Yaskawa INFORM job: FRONT_WELD_0ST-2_4640.JBI

/JOB
//NAME FRONT_WELD_0ST-2_4640
///FOLDERNAME 02-SKRZYNIE_JOBS
//POS
///NPOS 115,115,0,17,0,0
///TOOL 0
///POSTYPE PULSE
///PULSE
C00000=1212,-39190,49707,1936,-15809,-581
C00001=-55064,-17017,13106,20113,45767,-35735
C00002=-85641,-3161,12660,31281,67420,-55579
C00003=-77611,9747,38455,32702,57795,-55547
C00004=-77611,9747,38455,32702,57795,-55547
C00005=-80481,23547,61641,37204,60115,-56891
C00006=-80479,11681,28780,33754,71138,-52780
C00007=-73572,15026,34389,33675,67405,-51294
C00008=-73572,19926,48501,35202,62492,-53068
C00009=-82806,26311,53816,38180,73291,-53604
C00010=-71695,3747,16001,30713,64750,-51022
C00011=-70421,5575,20105,30867,63066,-51036
C00012=-35543,-20105,-5144,22821,50284,-40173
C00013=-37830,-23193,-8618,23571,50957,-40982
C00014=11136,-28839,-12562,1025,41780,-20887
C00015=20486,-27077,-7346,-12554,38415,-10736
C00016=59545,-9921,5571,-27063,51925,3267
C00017=55110,-17412,-5825,-19778,50988,-2825
C00018=79390,11759,28162,-35512,71262,52960
C00019=74811,13878,33986,-35807,67493,52464
C00020=74942,18762,48004,-37392,62815,54352
C00021=76815,18630,46530,-37158,64288,54543
C00022=79390,11759,28162,-35512,71262,52960
C00023=10831,-54278,-29128,-6468,39852,-5090
C00024=-67200,-10549,24402,-3189,24913,-39001
C00025=-75122,-2194,12822,3152,39225,-43427
C00026=-77516,10189,32861,8493,33365,-45533
C00027=-75154,17575,49272,7885,27457,-44928
C00028=-68113,9932,38901,1157,28472,-40453
C00029=-67114,5383,31515,9208,32648,-43213
C00030=-66450,3998,29285,10896,33890,-43630
C00031=-66374,3101,28136,14657,35566,-44954
C00032=-66747,-26,23691,26916,43760,-49061
C00033=-69992,3685,29239,35234,50920,-52492
C00034=-77050,-3138,8526,33226,61087,-51698
C00035=-67200,-10549,24402,-3189,24913,-39001
C00036=0,-52280,40443,83103,28146,-16510
C00037=99993,-20782,22705,-13349,24734,56519
C00038=67200,-10549,24402,3189,24913,39001
C00039=75122,-2194,12822,-3152,39225,43427
C00040=74323,5203,27259,-5972,33194,43789
C00041=74015,16414,48063,-6821,27325,44224
C00042=56519,1138,28747,9235,29393,33453
C00043=55467,619,28251,10155,29461,32830
C00044=56374,-724,25854,4078,30541,35419
C00045=56354,-7060,16047,-17622,38436,43274
C00046=68252,956,25699,-34035,49810,51639
C00047=77050,-3138,8526,-33226,61087,51698
C00048=67200,-10549,24402,3189,24913,39001
C00049=0,-52280,40443,-83103,28146,16510
C00050=-99993,-20782,22705,13349,24734,-56519
C00051=-91125,453,39555,30378,52425,-51131
C00052=-81425,-5449,14825,37552,56592,-47667
C00053=-81425,-10835,-2515,34915,62871,-45127
C00054=-79239,4305,16082,37593,68846,-50182
C00055=-81302,5892,27588,46359,62943,-54679
C00056=-82227,19402,59913,51524,57300,-60581
C00057=-84844,8890,27031,38640,69740,-53449
C00058=-90096,4679,14083,37467,76581,-51973
C00059=-87885,29238,52923,40761,81198,69685
C00060=-84355,23847,39024,40698,83720,72224
C00061=-81960,27335,46957,41070,80536,71891
C00062=-82643,24718,50492,48951,72637,70260
C00063=-90480,18737,31939,47254,81986,71631
C00064=-94217,10634,17426,46901,86469,-59967
C00065=-81425,-10835,-2515,34915,62871,-45127
C00066=-81425,-5449,14825,37552,56592,-47667
C00067=-94290,-610,44819,32366,49686,-53459
C00068=0,-55136,17047,60468,32096,-4233
C00069=99993,-20782,22705,-13349,24734,56519
C00070=91125,453,39555,-30378,52425,51131
C00071=81425,-5449,14825,-37552,56592,47667
C00072=81425,-10835,-2515,-34915,62871,45127
C00073=79239,4305,16082,-37593,68846,50182
C00074=83239,4964,30263,-50637,62037,57149
C00075=83991,16425,61235,-57769,55250,63273
C00076=93928,7973,40920,-53095,64494,61640
C00077=75109,22299,39152,-26915,78743,47998
C00078=79256,17348,34699,-33448,76412,88212
C00079=79932,23608,50901,-39863,71219,88955
C00080=76220,30771,63034,-41386,67395,88927
C00081=86322,16060,37848,-39554,76452,89287
C00082=87424,-1569,9538,-38190,72401,52253
C00083=81425,-10835,-2515,-34915,62871,45127
C00084=92850,-11266,9233,-39092,60986,50964
C00085=28366,-40369,19479,-5635,23506,17663
C00086=-80334,-19501,31260,21216,42469,-40219
C00087=-80621,-32280,-9061,25825,59412,-41877
C00088=-80621,-37319,-22868,24573,64555,-40576
C00089=-75108,-2453,16462,35304,60348,-42510
C00090=-72509,6961,33136,36537,55809,-43202
C00091=-35516,-19804,6201,28214,41034,-31537
C00092=-39606,-22901,-1163,28356,44724,-32188
C00093=15344,-29112,-5358,-2858,33820,-6852
C00094=13899,-24312,2834,-1929,31756,-7563
C00095=57847,-8680,15920,-27181,42395,12892
C00096=60973,-17187,4937,-27817,44388,13718
C00097=60973,-17187,4937,-27817,44388,13718
C00098=-13287,-42463,-12044,19170,31021,-23010
C00099=-17374,-21287,20534,22794,29118,-26096
C00100=13276,-20759,18622,-1911,29377,-7028
C00101=39924,-14247,19329,-14795,35999,4396
C00102=41528,-14133,18797,-15449,36702,5040
C00103=57001,-5890,26499,-21893,40771,11494
C00104=64054,-19541,3059,-29141,44956,15011
C00105=51466,-33957,-1499,-46586,51805,23434
C00106=17032,-20770,22044,-28854,30468,11088
C00107=-9868,-18638,14971,-8492,38486,-5199
C00108=-40562,-13194,19800,9508,35447,-20184
C00109=-41848,-12620,20103,10165,35810,-20773
C00110=-57278,-4046,28217,17578,39066,-27653
C00111=-71680,-19835,10874,33863,39440,-36917
C00112=-20806,-37586,-12792,9951,42782,-18031
///LIMIT ON
C00113=29087,-45372,27330,-13325,19529,9021
C00114=0,-35121,73515,0,-2982,0
///LIMIT OFF
BC00000=771029
BC00001=822981
BC00002=826240
BC00003=826240
BC00004=826240
BC00005=826240
BC00006=843102
BC00007=843104
BC00008=843104
BC00009=843104
BC00010=843104
BC00011=843104
BC00012=843104
BC00013=843104
BC00014=843104
BC00015=843103
BC00016=843104
BC00017=843105
BC00018=843105
BC00019=843105
BC00020=843105
BC00021=843105
BC00022=843105
BC00023=838615
BC00024=814763
BC00025=843940
BC00026=843943
BC00027=843943
BC00028=843940
BC00029=843941
BC00030=843942
BC00031=843942
BC00032=843943
BC00033=843943
BC00034=843943
BC00035=814763
BC00036=743369
BC00037=743369
BC00038=814763
BC00039=843940
BC00040=843943
BC00041=843943
BC00042=843943
BC00043=843943
BC00044=843948
BC00045=843955
BC00046=843944
BC00047=843943
BC00048=814763
BC00049=743369
BC00050=743369
BC00051=780831
BC00052=826634
BC00053=846031
BC00054=846033
BC00055=846033
BC00056=846033
BC00057=846033
BC00058=846609
BC00059=846033
BC00060=859972
BC00061=859972
BC00062=859972
BC00063=859972
BC00064=859972
BC00065=846031
BC00066=826634
BC00067=780831
BC00068=781117
BC00069=743369
BC00070=780831
BC00071=826634
BC00072=846031
BC00073=846033
BC00074=846033
BC00075=846033
BC00076=846033
BC00077=846033
BC00078=846033
BC00079=846033
BC00080=846033
BC00081=846033
BC00082=846033
BC00083=846031
BC00084=826634
BC00085=757646
BC00086=772124
BC00087=791684
BC00088=829989
BC00089=829989
BC00090=829989
BC00091=829987
BC00092=829989
BC00093=829989
BC00094=829989
BC00095=829987
BC00096=829989
BC00097=822654
BC00098=829989
BC00099=829989
BC00100=829985
BC00101=829987
BC00102=830031
BC00103=829987
BC00104=829989
BC00105=829989
BC00106=829985
BC00107=829987
BC00108=829989
BC00109=829989
BC00110=829989
BC00111=829989
BC00112=826581
BC00113=713357
BC00114=605515
///POSTYPE BASE
///RECTAN
///RCONF 0,0,0,0,0,0,0,0,0,0,0,0,0,0,0,0,0,0,0,0,0,0,0,0
P00021=6.550,-0.003,-5.735,0.0000,0.0000,0.0000
P00022=5.943,-0.018,-6.388,0.0000,0.0000,0.0000
P00023=7.025,-0.019,-7.168,0.0000,0.0000,0.0000
P00024=5.926,-0.047,-4.777,0.0000,0.0000,0.0000
P00350=11.519,-0.008,1.149,0.0000,0.0000,0.0000
P00351=13.563,-0.027,-0.653,0.0000,0.0000,0.0000
P00352=13.252,-0.027,-0.827,0.0000,0.0000,0.0000
P00353=10.971,-0.082,0.776,0.0000,0.0000,0.0000
P00399=-2.449,0.031,8.825,0.0000,0.0000,0.0000
P00400=5.920,-3.503,-0.024,0.0000,0.0000,0.0000
P00401=3.430,-0.021,1.131,0.0000,0.0000,0.0000
P00402=-0.253,1.107,3.062,0.0000,0.0000,0.0000
P00403=-3.666,-0.015,5.328,0.0000,0.0000,0.0000
P00405=2.420,0.007,1.427,0.0000,0.0000,0.0000
P00406=3.513,-0.022,0.429,0.0000,0.0000,0.0000
P00415=-1.781,-1.303,3.250,0.0000,0.0000,0.0000
P00416=0.027,1.119,3.078,0.0000,0.0000,0.0000
//INST
///DATE 2024/06/25 12:05
///ATTR SC,RW
///GROUP1 RB1,BS1
NOP
'**********************
'**********************
'POCZATEK SPAWANIA PRZOD
'**********************
'**********************
MOVJ C00000 BC00000 VJ=60.00
MOVL C00001 BC00001 V=416.7
MOVJ C00002 BC00002 VJ=10.00
MOVJ C00003 BC00003 VJ=10.00
MOVL C00004 BC00004 V=150.0
MOVL C00005 BC00005 V=150.0
'**********************
'W41A SIDE
'**********************
MOVL C00006 BC00006 V=250.0
SFTON P0402
MOVL C00007 BC00007 V=66.7 PL=0
MACRO1 MJ#(0) ARGF14
ARCON
MOVL C00008 BC00008 V=9.2
ARCOF
SFTOF
MOVL C00009 BC00009 V=166.7
'**********************
'W41A FRONT
'**********************
MOVL C00010 BC00010 V=250.0
SFTON P0350
MOVL C00011 BC00011 V=66.7 PL=0
SFTOF
MACRO1 MJ#(0) ARGF21
ARCON
SFTON P0351
MOVL C00012 BC00012 V=8.3
SFTOF
ARCOF
MOVL C00013 BC00013 V=166.7
'**********************
'W41B FRONT
'**********************
MOVL C00014 BC00014 V=250.0
SFTON P0352
MOVL C00015 BC00015 V=66.7 PL=0
SFTOF
MACRO1 MJ#(0) ARGF21
ARCON
SFTON P0353
MOVL C00016 BC00016 V=8.3
SFTOF
ARCOF
MOVL C00017 BC00017 V=166.7
MOVL C00018 BC00018 V=100.0
'**********************
'W41A SIDE
'**********************
SFTON P0400
MOVL C00019 BC00019 V=66.7 PL=0
MACRO1 MJ#(0) ARGF21
ARCON
MOVL C00020 BC00020 V=8.3
ARCOF
SFTOF
MOVL C00021 BC00021 V=166.7
MOVL C00022 BC00022 V=166.7
MOVL C00023 BC00023 V=333.3
MOVJ C00024 BC00024 VJ=20.00
MOVJ C00025 BC00025 VJ=20.00
'**********************
'W42A.1
'**********************
'POPRAWIC
MOVL C00026 BC00026 V=500.0
SFTON P0403
MOVL C00027 BC00027 V=66.7 PL=0
MACRO1 MJ#(0) ARGF9
ARCON
MOVL C00028 BC00028 V=9.2
SFTON P0416
MOVL C00029 BC00029 V=9.2
MOVL C00030 BC00030 V=9.2
MOVL C00031 BC00031 V=9.2
SFTON P0402
MOVL C00032 BC00032 V=9.2
MOVL C00033 BC00033 V=9.2
ARCOF
MOVL C00034 BC00034 V=500.0
SFTOF
MOVJ C00035 BC00035 VJ=15.00
'W42B.1
MOVJ C00036 BC00036 VJ=30.00
MOVJ C00037 BC00037 VJ=30.00
MOVJ C00038 BC00038 VJ=30.00
MOVJ C00039 BC00039 VJ=30.00
'**********************
'W42B.1
'**********************
MOVL C00040 BC00040 V=500.0
SFTON P0399
MOVL C00041 BC00041 V=166.7 PL=0
MACRO1 MJ#(0) ARGF9
ARCON
SFTON P0415
MOVL C00042 BC00042 V=9.2
MOVL C00043 BC00043 V=9.2
MOVL C00044 BC00044 V=9.2
SFTON P0400
MOVL C00045 BC00045 V=9.2
MOVL C00046 BC00046 V=9.2
ARCOF
MOVL C00047 BC00047 V=500.0
SFTOF
MOVJ C00048 BC00048 VJ=25.00
'W42A.2
MOVJ C00049 BC00049 VJ=40.00
MOVJ C00050 BC00050 VJ=30.00
MOVJ C00051 BC00051 VJ=30.00
MOVJ C00052 BC00052 VJ=30.00
MOVJ C00053 BC00053 VJ=30.00
'**********************
'W42A.2
'**********************
MOVL C00054 BC00054 V=500.0
SFTON P0402
MOVL C00055 BC00055 V=166.7 PL=0
SFTOF
MACRO1 MJ#(0) ARGF9
ARCON
SFTON P0402
MOVL C00056 BC00056 V=9.2
ARCOF
MOVL C00057 BC00057 V=166.7
MOVJ C00058 BC00058 VJ=20.00
MOVJ C00059 BC00059 VJ=20.00
MOVL C00060 BC00060 V=250.0
MOVL C00061 BC00061 V=166.7
ARCON
MOVL C00062 BC00062 V=10.8
ARCOF
MOVL C00063 BC00063 V=166.7
MOVJ C00064 BC00064 VJ=20.00
SFTOF
MOVJ C00065 BC00065 VJ=30.00
MOVJ C00066 BC00066 VJ=30.00
MOVJ C00067 BC00067 VJ=30.00
'W42B.2
MOVJ C00068 BC00068 VJ=30.00
MOVJ C00069 BC00069 VJ=30.00
MOVJ C00070 BC00070 VJ=30.00
MOVJ C00071 BC00071 VJ=30.00
MOVJ C00072 BC00072 VJ=30.00
'**********************
'W42B.2
'**********************
MOVL C00073 BC00073 V=500.0
SFTON P0400
MOVL C00074 BC00074 V=166.7 PL=0
SFTOF
MACRO1 MJ#(0) ARGF9
ARCON
SFTON P0400
MOVL C00075 BC00075 V=9.2
ARCOF
SFTOF
MOVL C00076 BC00076 V=250.0
MOVL C00077 BC00077 V=166.7
MOVJ C00078 BC00078 VJ=10.00
SFTON P0400
MOVL C00079 BC00079 V=166.7
ARCON
MOVL C00080 BC00080 V=10.8
ARCOF
MOVL C00081 BC00081 V=250.0
MOVL C00082 BC00082 V=500.0
SFTOF
MOVJ C00083 BC00083 VJ=20.00
MOVJ C00084 BC00084 VJ=30.00
'W42A.3
MOVJ C00085 BC00085 VJ=20.00
MOVJ C00086 BC00086 VJ=20.00
MOVJ C00087 BC00087 VJ=30.00
MOVJ C00088 BC00088 VJ=30.00
'**********************
'W42A.3
'**********************
MOVL C00089 BC00089 V=500.0
SFTON P0021
MOVL C00090 BC00090 V=166.7 PL=0
MACRO1 MJ#(0) ARGF9
ARCON
SFTON P0022
MOVL C00091 BC00091 V=9.2
ARCOF
MOVL C00092 BC00092 V=500.0
SFTOF
'**********************
'W42B.3
'**********************
MOVL C00093 BC00093 V=500.0
SFTON P0023
MOVL C00094 BC00094 V=166.7 PL=0
ARCON
SFTON P0024
MOVL C00095 BC00095 V=9.2
ARCOF
MOVL C00096 BC00096 V=500.0
SFTOF
MOVJ C00097 BC00097 VJ=20.00
'**********************
'GORA L
'**********************
MOVL C00098 BC00098 V=500.0
SFTON P0401
MOVL C00099 BC00099 V=166.7 PL=0
MACRO1 MJ#(0) ARGF9
ARCON
MOVL C00100 BC00100 V=11.7
SFTON P0406
MOVL C00101 BC00101 V=11.7
MOVL C00102 BC00102 V=11.7
MOVL C00103 BC00103 V=11.7
ARCOF
MOVL C00104 BC00104 V=500.0
SFTOF
'**********************
'GORA P
'**********************
MOVL C00105 BC00105 V=166.7
SFTON P0401
MOVL C00106 BC00106 V=166.7 PL=0
ARCON
MOVL C00107 BC00107 V=11.7
SFTON P0405
MOVL C00108 BC00108 V=11.7
MOVL C00109 BC00109 V=11.7
MOVL C00110 BC00110 V=11.7
ARCOF
MOVL C00111 BC00111 V=500.0
SFTOF
MOVJ C00112 BC00112 VJ=20.00
MOVJ C00113 BC00113 VJ=30.00
MOVJ C00114 BC00114 VJ=30.00
'KONIEC SPAWANIA FRONTU
END
